FUNCTION_BLOCK Switch EXTENDS Axis_Base IMPLEMENTS I_Lift
VAR
	_Assigned : BOOL;
END_VAR

PROPERTY Assigned : BOOL
GET
Assigned := _Assigned;
END_GET
SET
_Assigned := Assigned;
END_SET
END_PROPERTY

METHOD Call : HRESULT
VAR_INPUT
	Position : LREAL;
	Velocity : LREAL;
END_VAR
IF Assigned THEN
	RETURN;
	Call := -1;
END_IF

Call := (MoveToModuloPosition(Position := Position, Velocity := Velocity));
END_METHOD

METHOD Release : HRESULT
VAR_INPUT
END_VAR
_Assigned := FALSE;
END_METHOD

END_FUNCTION_BLOCK

(* stored: Version 1.1.0.1
   POU Switch: Id {074ec01d-efeb-40bf-b31f-8bc7084e0e0c}, SpecialFunc None
   Property Assigned: Id {fe993b0e-f1e9-419b-83a4-8730860a9e18}
   Get Get: Id {5abe71d0-8308-4f05-9fc2-3c34e26d1741}
   Set Set: Id {acc098ff-5872-48dc-b763-c9d1fb7af925}
   Method Call: Id {58c6f245-50e0-4e4b-a8ae-1bc1d34e6a27}
   Method Release: Id {daad8677-99cd-44be-bf6a-0aa91a7d9e5d} *)
